# EPICS autosave request: iocBoot/obsolete/ioc13Galil_test/auto_positions.req
file "CARS_8_motor_positions.req",         P=$(P)
~
